(* IEC 61131-3 sources: POMIRTS_lab3/AS/Library_2/ArSsl, 3 files *)

(* ---- ArSsl.typ ---- *)
TYPE
	ArSslCipherVersionEnum :
		(
            arSSL_SSL_3_0 := 1,				(*SSL 3.0*) (**) (*#PAR*)
			arSSL_TLS_1_0 := 2				(*TLS 1.0*) (**) (*#PAR*)
        );

	ArSslCfgOwnCertificateType : STRUCT
		Certificate		: STRING[255]; 			(*name of the own certificate*) (**) (*#PAR*)
		PrivateKey		: STRING[255]; 			(*name of the private key of the own certificate*) (**) (*#PAR*)
		Password		: STRING[255];			(*password of the private key*) 	(**) (*#PAR*)
	END_STRUCT;

	ArSslCfgOwnCertDetailsType : STRUCT
		Certificate		: STRING[255]; 			(*name of the own certificate*) (**) (*#PAR*)
		PrivateKey		: STRING[255]; 			(*name of the private key of the own certificate*) (**) (*#PAR*)
	END_STRUCT;

	ArSslCfgType : STRUCT		(*details of an SSL configuration*)
		OwnCertificate		: ArSslCfgOwnCertificateType; 	(*the own certificate*) (**) (*#PAR*)
		SslVersion		: ArSslCipherVersionEnum;	(*SSL version*)		 	(**) (*#PAR*)
		TrustedCertificates 	: UDINT;			(*pointer to the trusted certificates (given as pointer to ARRAY OF STRING[255]) *)
		TrustedCertificateCount	: UDINT;			(*number of trusted certificates*)
		CRLs	 		: UDINT;			(*pointer to the certificate revocation lists (given as pointer to ARRAY OF STRING[255]) *) 	(**) (*#PAR*)
		CRLCount		: UDINT;			(*number of certificate revocation lists*) 	(**) (*#PAR*)
	END_STRUCT;

	ArSslCfgDetailsType : STRUCT	(*details of an SSL configuration*)
		Name				: STRING[255];			(*name of the SSL configuration*)
		OwnCertificate		: ArSslCfgOwnCertDetailsType; 	(*name of the own certificate*) (**) (*#PAR*)
		SslVersion			: ArSslCipherVersionEnum;	(*SSL cipher version*)		 	(**) (*#PAR*)
		CipherCount			: UDINT;			(*number of ciphers*)	(**) (*#PAR*)
		TrustedCertificateCount		: UDINT;			(*number of trusted certificates*)	(**) (*#PAR*)
		CRLCount 			: UDINT;			(*number of CRLs*) 	(**) (*#PAR*)
	END_STRUCT;

	ArSslAsyncInternalType : STRUCT
		FBStateCtx		: ArFBStateInternalType;
		AsyFuMaCtx		: ArFBAsyFuMaInternalType;
	END_STRUCT;
END_TYPE

(* ---- ArSsl.var ---- *)
VAR CONSTANT
	arSSL_ERR_CRLS_INVALID             : DINT := -1070585996;    (*invalid given; CRLs can only be used with trusted certificates*)
	arSSL_ERR_IDENT_INVALID            : DINT := -1070585995;    (*invalid identifier specified*)
	arSSL_ERR_SSL_CFG_NOT_FOUND        : DINT := -1070585994;    (*SSL configuration not found*)
	arSSL_ERR_CERTIFICATE_INVALID      : DINT := -1070585993;    (*invalid certificate given*)
	arSSL_ERR_PRIVATE_KEY_NOT_FOUND    : DINT := -1070585992;    (*private key not found*)
	arSSL_ERR_PASSWORD_INVALID         : DINT := -1070585991;    (*invalid password given*)
	arSSL_ERR_INTERNAL                 : DINT := -1070585990;    (*internal error*)
	arSSL_ERR_INDEX_OUT_OF_RANGE       : DINT := -1070585989;    (*given index is out of range*)
	arSSL_ERR_CFG_ALREADY_EXISTS       : DINT := -1070585988;    (*given SSL configuration already exists*)
	arSSL_ERR_NAME_INVALID             : DINT := -1070585987;    (*invalid name given*)
	arSSL_ERR_OWN_CERT_INVALID         : DINT := -1070585986;    (*invalid own certificate given*)
	arSSL_ERR_PRIVATE_KEY_INVALID      : DINT := -1070585985;    (*invalid own private key given*)
	arSSL_ERR_SSL_VERSION_INVALID      : DINT := -1070585984;    (*invalid SSL version given*)
	arSSL_ERR_TRUSTED_DATA_INVALID     : DINT := -1070585983;    (*invalid trusted data given*)
	arSSL_ERR_TRUSTEDCOUNT_INVALID     : DINT := -1070585982;    (*invalid trusted count given*)
	arSSL_ERR_CRLS_DATA_INVALID        : DINT := -1070585981;    (*invalid CRLs data given*)
	arSSL_ERR_CRLCOUNT_INVALID         : DINT := -1070585980;    (*invalid CRL count given*)
END_VAR

(* ---- ArSsl.fun ---- *)
{REDUND_CONTEXT} {REDUND_UNREPLICABLE} FUNCTION_BLOCK ArSslCreateCfg   					(*creates an SSL configuration entry*)
	VAR_INPUT
		Execute			: BOOL; 			(*starts execution*) 				(**) (*#PAR*)
		Name 			: STRING[255];			(*name of the SSL configuration*) 	(**) (*#PAR*)
		Configuration		: ArSslCfgType;			(*configuration settings of an SSL configuration*) 	(**) (*#PAR*)
	END_VAR
	VAR_OUTPUT
		Done			: BOOL;				(*execution done*) 				(**) (*#PAR*)
		Busy			: BOOL;				(*execution running*) 			(**) (*#PAR*)
		Error			: BOOL;				(*execution failed*) 			(**) (*#PAR*)
		StatusID		: DINT;  			(*execution error: see help*) 	(**) (*#PAR*)
	END_VAR
	VAR
		Internal		: ArSslAsyncInternalType;	(*interne Variable*)
	END_VAR
END_FUNCTION_BLOCK

{REDUND_CONTEXT} {REDUND_UNREPLICABLE} FUNCTION_BLOCK ArSslDeleteCfg		   				(*deletes an existing SSL configuration entry*)
	VAR_INPUT
		Execute			: BOOL; 			(*starts execution*) 				(**) (*#PAR*)
		Name			: STRING[255];			(*name of the SSL configuration*) 	(**) (*#PAR*)
	END_VAR
	VAR_OUTPUT
		Done			: BOOL;				(*execution done*) 				(**) (*#PAR*)
		Busy			: BOOL;				(*execution running*) 			(**) (*#PAR*)
		Error			: BOOL;				(*execution failed*) 			(**) (*#PAR*)
		StatusID		: DINT;  			(*execution error: see help*) 	(**) (*#PAR*)
	END_VAR
	VAR
		Internal		: ArSslAsyncInternalType;	(*internal variable*)
	END_VAR
END_FUNCTION_BLOCK

{REDUND_CONTEXT} {REDUND_UNREPLICABLE} FUNCTION_BLOCK ArSslOpen   		   				(*opens an existing SSL configuration*)
	VAR_INPUT
		Execute			: BOOL; 			(*starts execution*) 			(**) (*#PAR*)
		Name 			: STRING[255];			(*name of the SSL configuration*) 	(**) (*#PAR*)
	END_VAR
	VAR_OUTPUT
		Ident			: UDINT;			(*identifier of the SSL configuration*)
		Done			: BOOL;				(*execution done*) 				(**) (*#PAR*)
		Busy			: BOOL;				(*execution running*) 			(**) (*#PAR*)
		Error			: BOOL;				(*execution failed*) 			(**) (*#PAR*)
		StatusID		: DINT;  			(*execution error: see help*) 	(**) (*#PAR*)
	END_VAR
	VAR
		Internal		: ArSslAsyncInternalType;	(*internal variable*)
	END_VAR
END_FUNCTION_BLOCK

{REDUND_CONTEXT} {REDUND_UNREPLICABLE} FUNCTION_BLOCK ArSslClose 	    					(*closes an existing SSL configuration*)
	VAR_INPUT
		Ident			: UDINT;			(*identifier of the SSL configuration*)
		Execute			: BOOL; 			(*starts execution*) 			(**) (*#PAR*)
	END_VAR
	VAR_OUTPUT
		Done			: BOOL;				(*execution done*) 				(**) (*#PAR*)
		Busy			: BOOL;				(*execution running*) 			(**) (*#PAR*)
		Error			: BOOL;				(*execution failed*) 			(**) (*#PAR*)
		StatusID		: DINT;  			(*execution error: see help*) 	(**) (*#PAR*)
	END_VAR
	VAR
		Internal		: ArSslAsyncInternalType;	(*internal variable*)
	END_VAR
END_FUNCTION_BLOCK

{REDUND_CONTEXT} {REDUND_UNREPLICABLE} FUNCTION_BLOCK ArSslGetCfgDetails					(*gets details from an SSL configuration*)
	VAR_INPUT
		Execute			: BOOL; 			(*starts execution*) 			(**) (*#PAR*)
		Name 			: STRING[255];			(*name of the SSL configuration*)	(**) (*#PAR*)
		Index			: UDINT;			(*index of the SSL configuration*) (**) (*#PAR*)
	END_VAR
	VAR_OUTPUT
		Done			: BOOL;				(*execution done*) 				(**) (*#PAR*)
		Busy			: BOOL;				(*execution running*) 			(**) (*#PAR*)
		Error			: BOOL;				(*execution failed*) 			(**) (*#PAR*)
		StatusID		: DINT;  			(*execution error: see help*) 	(**) (*#PAR*)
		Details			: ArSslCfgDetailsType;		(*details of an SSL configuration*) 	(**) (*#PAR*)
	END_VAR
	VAR
		Internal		: ArSslAsyncInternalType;	(*internal variable*)
	END_VAR
END_FUNCTION_BLOCK

{REDUND_CONTEXT} {REDUND_UNREPLICABLE} FUNCTION_BLOCK ArSslGetCipher 						(*gets the cipher with given index of the given SSL configuration*)
	VAR_INPUT
		Execute			: BOOL; 			(*starts execution*) 			(**) (*#PAR*)
		Name 			: STRING[255];			(*name of the SSL configuration*) 	(**) (*#PAR*)
		Index			: UDINT;			(*index of the cipher*) (**) (*#PAR*)
	END_VAR
	VAR_OUTPUT
		Done			: BOOL;				(*execution done*) 				(**) (*#PAR*)
		Busy			: BOOL;				(*execution running*) 			(**) (*#PAR*)
		Error			: BOOL;				(*execution failed*) 			(**) (*#PAR*)
		StatusID		: DINT;  			(*execution error: see help*) 	(**) (*#PAR*)
		Cipher			: STRING[63];			(*cipher*) 	(**) (*#CMD*)
	END_VAR
	VAR
		Internal		: ArSslAsyncInternalType;	(*interne Variable*)
	END_VAR
END_FUNCTION_BLOCK

{REDUND_CONTEXT} {REDUND_UNREPLICABLE} FUNCTION_BLOCK ArSslGetCertificate 					(*gets the trusted certificate with given index of the given SSL configuration*)
	VAR_INPUT
		Execute			: BOOL; 			(*starts execution*) 			(**) (*#PAR*)
		Name 			: STRING[255];			(*name of the SSL configuration*) 	(**) (*#PAR*)
		Index			: UDINT;			(*index of the trusted certificate*) (**) (*#PAR*)
	END_VAR
	VAR_OUTPUT
		Done			: BOOL;				(*execution done*) 				(**) (*#PAR*)
		Busy			: BOOL;				(*execution running*) 			(**) (*#PAR*)
		Error			: BOOL;				(*execution failed*) 			(**) (*#PAR*)
		StatusID		: DINT;  			(*execution error: see help*) 	(**) (*#PAR*)
		TrustedCertificate	: STRING[255];			(*trusted certificate*) 	(**) (*#CMD*)
	END_VAR
	VAR
		Internal		: ArSslAsyncInternalType;	(*interne Variable*)
	END_VAR
END_FUNCTION_BLOCK

{REDUND_CONTEXT} {REDUND_UNREPLICABLE} FUNCTION_BLOCK ArSslGetCRL 					(*gets the certificate revocation list with given index of the given SSL configuration*)
	VAR_INPUT
		Execute			: BOOL; 			(*starts execution*) 			(**) (*#PAR*)
		Name 			: STRING[255];			(*name of the SSL configuration*) 	(**) (*#PAR*)
		Index			: UDINT;			(*index of the trusted certificate*) (**) (*#PAR*)
	END_VAR
	VAR_OUTPUT
		Done			: BOOL;				(*execution done*) 				(**) (*#PAR*)
		Busy			: BOOL;				(*execution running*) 			(**) (*#PAR*)
		Error			: BOOL;				(*execution failed*) 			(**) (*#PAR*)
		StatusID		: DINT;  			(*execution error: see help*) 	(**) (*#PAR*)
		CRL			: STRING[255];			(*certificate revocation list*) 	(**) (*#CMD*)
	END_VAR
	VAR
		Internal		: ArSslAsyncInternalType;	(*interne Variable*)
	END_VAR
END_FUNCTION_BLOCK
